SYMBOL_TABLE
"CONTROL_DAT"	DB 1	DB 1
"MODBUS_HPARAM_PN_2"	DB 2	DB 2
"CPULINDB"	DB 30	DB 30
"SYS_Date_Time_D"	DB 34	DB 34	// 系统日期和时间设置和读取数据区
"FB200_DB"	DB 200	FB 200
"FB201_DB"	DB 201	FB 201
"MAIN-READ-SLAVE"	DB 202	DB 202
"MAIN-WRITE-SLAVE"	DB 203	DB 203
"MAIN-READ-IBP"	DB 204	DB 204
"MAIN-WRITE-IBP"	DB 205	DB 205
"DETAIL_DIAG_DB_RACK0"	DB 458	FB 315	// DB FOR SFB13
"DETAIL_DIAG_DB_RACK1"	DB 459	FB 315	// DB FOR SFB12
"DP_ERROR_RACK0"	DB 460	DB 460
"DP_ERROR_RESET_DB"	DB 461	DB 461
"DP_ERROR_FB1501"	DB 462	FB 1501
"DB_FOR_FB300"	DB 463	FB 300
"DP_VAT"	DB 464	DB 464
"DP_ERROR_RACK1"	DB 465	DB 465
"DP_ERROR1_RESET"	DB 466	DB 466
"DP_ERROR1_FB1501"	DB 467	FB 1501
"FB523_DB"	DB 523	FB 523
"LED"	DB 525	DB 525
"IDB_MODBUS"	DB 915	FB 915
"JOBLIST_DB"	DB 919	FB 919
"JOB_RESET_DB"	DB 921	FB 921
"LSQK-1"	DB 2005	DB 2005
"EPS22"	DB 2015	DB 2015
"AP-PSB"	DB 2025	DB 2025
"XFSW"	DB 2035	DB 2035
"ZNZM_WRITE"	DB 2053	DB 2053
"ZNZM_READ"	DB 2055	DB 2055
"YSB_1_2"	DB 2065	DB 2065
"YSB_3_4"	DB 2075	DB 2075
"AP PSB  WSB"	DB 2115	DB 2115
"E420/04(K1)"	DB 2125	DB 2125
"E420/08(K4)"	DB 2135	DB 2135
"H420/02(K4)"	DB 2145	DB 2145
"E402\02_N RE"	DB 2185	DB 2185
"IMCC_Read"	DB 2291	DB 2291	// IMCC系统读取数据
"IMCC_Write"	DB 2292	DB 2292	// IMCC系统写数据
"HF3_EPS_HMI"	DB 2501	FB 2501	// EPS_ToHMI
"IMCC_lock"	DB 2555	DB 2555
"MAIN_HMI_SCtrl"	DB 6001	DB 6001	// HMI控制设备DB
"MAIN_ToHMI"	DB 6002	DB 6002	// 发送数据至HMI
"SLAVE_HMI_SCtrl"	DB 6003	DB 6003
"SLAVE_ToHMI"	DB 6004	DB 6004
"IBP_HMI_SCtrl"	DB 6005	DB 6005
"IBP_ToHMI"	DB 6006	DB 6006
"HF3_DP_Statu_ToHMI"	DB 6007	DB 6007
"HF3_PLC_Statu_ToHMI"	DB 6008	DB 6008
"HF4_Sum_SCtrl"	DB 6040	DB 6040
"HF3_Mode_Table"	DB 7001	DB 7001	// 下载模式总表
"HF3_Act_Mode"	DB 7002	DB 7002
"HF3_Init_Mode_Index"	DB 7003	DB 7003	// 系统模式分区索引
"HF3_Mode_DB"	DB 7004	DB 7004	// 模式内部使用DB
"Maste_To_Slave_Mod_DB"	DB 7005	DB 7005	// 从端反馈模式信息至主端
"HF3_Slave_To_Maste_Mode"	DB 7006	DB 7006	// 从端反馈模式状态
"P_RCV"	FB 12	FB 12	// Receive Data from CP340
"P_SEND"	FB 13	FB 13	// Send Data to CP340
"pid"	FB 41	FB 41
"TSEND"	FB 63	FB 63	// Send Data
"TRCV"	FB 64	FB 64	// Receive Data
"TCON"	FB 65	FB 65	// Connect
"TDISCON"	FB 66	FB 66	// Disconnect
"P_RESET"	FB 177	FB 177	// Reset Job for CP340
"S7400H-COM-MAIN-SLAVE"	FB 200	FB 200
"S7400H-COM-MAIN-IBP"	FB 201	FB 201
"READ_ERROR"	FB 300	FB 300
"DETAIL_DP_DIAG"	FB 315	FB 315
"H_STATUS"	FB 523	FB 523	// Status H-System
"HF3_ZNZM_Luxtrans"	FB 730	FB 730	// 智能照明照度转换
"TCP_COMM"	FB 913	FB 913	// TCP Kommunikation
"MOD_CLI"	FB 914	FB 914
"MB_PNHCL"	FB 915	FB 915
"Job_List"	FB 919	FB 919
"JOB_RESET"	FB 921	FB 921
"MODMAS_STEP7_CP340_L"	FB 1071	FB 1071
"com_check"	FB 1501	FB 1501
"HF3_PID_FB2005"	FB 2005	FB 2005	// PID处理功能块
"HF3_RunFaultSum"	FB 2006	FB 2006	// 运行时间故障次数统计
"HF3_EPS_FB2501"	FB 2501	FB 2501	// EPS主程序段
"HF4_EPS_FB2502"	FB 2502	FB 2502	// EPS功能块
"HF3_IMCC_CommOK_FB2512"	FB 2512	FB 2512	// IMCC心跳
"HF3_IMCC_CommOK_FB2513"	FB 2513	FB 2513
"HF3_LSQK_FB2521"	FB 2521	FB 2521	// 冷水群控程序段
"HF4_LSQK_FB2522"	FB 2522	FB 2522	// LSQK功能块
"HF3_JET_FB2531"	FB 2531	FB 2531	// 射流风机主程序端
"HF3_JET_FB2532"	FB 2532	FB 2532	// 射流风机功能块
"HF3_VRV_FB2541"	FB 2541	FB 2541	// 多联体空调主程序段
"HF3_VRV_FB2542"	FB 2542	FB 2542	// 多联体空调程序端
"HF4_SB_FB2551"	FB 2551	FB 2551	// 带控制水泵程序段
"HF4_SB_FB2552"	FB 2552	FB 2552	// 带控制水泵功能块
"HF4_3#SB_FB2561"	FB 2561	FB 2561	// 洞口水泵主程序段
"HF4_3#SB_FB2562"	FB 2562	FB 2562	// 洞口水泵功能块
"HF4_JSJYB_FB2571"	FB 2571	FB 2571	// 变频给水加压泵
"HF4_JSJYB"	FB 2572	FB 2572
"HF4_WSB_FB2581"	FB 2581	FB 2581	// 污水密闭提升
"HF4_WSB_FB2582"	FB 2582	FB 2582
"HF4_PSB_FB2591"	FB 2591	FB 2591	// 局部排水泵主程序
"HF4_PSB_FB2592"	FB 2592	FB 2592	// 排水泵DB转换
"HF4_1#PSB"	FB 2601	FB 2601
"HF4_1#PSB_FB2602"	FB 2602	FB 2602
"HF4_DT_FB2621"	FB 2621	FB 2621	// 电梯
"HF4_DT_FB2622"	FB 2622	FB 2622	// 电梯
"HF4_FT_FB2631"	FB 2631	FB 2631	// 扶梯
"HF4_FT_FB2362"	FB 2632	FB 2632
"HF3_FAS_FB2641"	FB 2641	FB 2641	// FAS主程序
"HF3_FAS_FB2642"	FB 2642	FB 2642
"HF3_FAS_COMM"	FB 2643	FB 2643	// 与FAS通讯功能块
"HF4_IMCC_TVF_FB2651"	FB 2651	FB 2651	// 隧道风机主程序段
"HF4_IMCC_TVF_FB2652"	FB 2652	FB 2652	// 隧道风机功能块
"HF4_IMCC_UOF_FB2661"	FB 2661	FB 2661	// 排热风机主程序
"HF4_IMCC_UOF_FB2662"	FB 2662	FB 2662	// 排热风机功能块
"HF4_IMCC_KT_FB2671"	FB 2671	FB 2671	// 大空调主程序
"HF4_IMCC_KT_FB2672"	FB 2672	FB 2672	// 空调机组功能块
"HF4_IMCC_HPF_FB2681"	FB 2681	FB 2681	// IMCC_HPF_主程序
"HF4_IMCC_HPF_FB2682"	FB 2682	FB 2682	// IMCC_HPF功能块
"HF4_IMCC_FJ_FB2691"	FB 2691	FB 2691	// 智能低压小风机
"HF4_IMCC_FJ_FB2692"	FB 2692	FB 2692	// 智能低压小风机功能块
"HF4_IMCC_DT_FB2711"	FB 2711	FB 2711	// IMCC风量调节阀程序
"HF4_IMCC_DT_FB2712"	FB 2712	FB 2712	// IMCC风量调节阀块
"HF4_IMCC_D_FB2721"	FB 2721	FB 2721	// IMCC电动风阀主程序
"HF4_IMCC_D_FB2722"	FB 2722	FB 2722	// IMCC电动风阀功能块
"HF4_JH_YC_FB2731"	FB 2731	FB 2731	// 电子净化压差主程序
"HF4_DPH_FB2751"	FB 2751	FB 2751	// 二通阀主程序
"HF4_DPH_FB2752"	FB 2752	FB 2752	// 二通阀主程序
"picontrol"	FB 2753	FB 2753
"HF3_FJ_FB2761"	FB 2761	FB 2761	// 高架站风机主程序段
"HF3_FJ_FB2762"	FB 2762	FB 2762	// 高架站风机
"HF4_FJPG_FB2771"	FB 2771	FB 2771	// 风机盘管主程序段
"HF4_FJPG_FB2772"	FB 2772	FB 2772	// 风机盘管功能块
"HF4_XFDF_FB2781"	FB 2781	FB 2781	// 手电一体蝶阀程序段
"HF4_XVDF_FB2782"	FB 2782	FB 2782	// 手电一体蝶阀功能块
"HF4_EPS_WLE_FB2791"	FB 2791	FB 2791	// 区间疏散指示
"HF4_EPS_WLE_FB2792"	FB 2792	FB 2792	// 区间疏散指示功能块
"HF3_D_FB2801"	FB 2801	FB 2801	// 高架站风阀主程序
"HF3_D_FB2802"	FB 2802	FB 2802	// 高架站风阀功能块
"HF4_FHF_RFM_FB2811"	FB 2811	FB 2811	// 防火阀人防门
"HF4_Senor_FB2821"	FB 2821	FB 2821	// 传感器程序段
"HF4_Sensor_FB2822"	FB 2822	FB 2822	// 传感器功能块
"AB_IBP_Comm"	FB 2831	FB 2831
"ZNZM_6biao"	FB 2841	FB 2841
"HF3_WSB_FB2852"	FB 2852	FB 2852
"HF3_Mode_Pro"	FB 3000	FB 3000	// 模式表总程序
"HF4_Mode_CAL_FB3001"	FB 3001	FB 3001
"HF3_Mode LookUp_FB3002"	FB 3002	FB 3002	// 查总模式表
"HF3_Mode_BE_Judge_FB3003"	FB 3003	FB 3003
"HF3_Sys_Grp_FB3004"	FB 3004	FB 3004	// 系统群控及状态上传
"HF3_Mode_Explode_FB3005"	FB 3005	FB 3005	// 模式表分解
"HF3_Mode_Condition_3006"	FB 3006	FB 3006
"HF3_SYS_Init"	FB 3007	FB 3007	// 系统初始化
"HF3_Slave_To_Maste"	FB 3009	FB 3009
"HF3_Mode_Refuse_FB3010"	FB 3010	FB 3010	// 模式不符合判断
"HF3_Big_LookUp_FB3012"	FB 3012	FB 3012	// 查表子程序
"HF3_Tub_LookUp_FB3013"	FB 3013	FB 3013
"HF3_little_LookUp_FB3014"	FB 3014	FB 3014
"HF3_WG_Be_Judge_FB3015"	FB 3015	FB 3015	// 判断模式开始/结束/执行中
"HF3_Sys_Grp_FB3016"	FB 3016	FB 3016
"HF3_LittleSys_Grp_FB3017"	FB 3017	FB 3017
"HF3_Mode_Condition_3018"	FB 3018	FB 3018
"HF3_Mode_Explode_FB3019"	FB 3019	FB 3019
"SDT"	FB 4180	FB 4180
"BAS_CGQ"	FB 4251	FB 4251
"IMCC_Pro"	FC 1	FC 1	// 智能低压通信数据段
"HF3_B_T_W_FC51"	FC 51	FC 51	// BOOLתWORD
"HF3_W_T_B_FC54"	FC 54	FC 54	// WORDתBOOL
"HF3_Bite_T_Bool_FC55"	FC 55	FC 55
"SCALE"	FC 105	FC 105	// Scaling Values
"UNSCALE"	FC 106	FC 106	// Unscaling Values
"MK_ERROR_SAVE_RACK0"	FC 201	FC 201
"RIO_Information"	FC 202	FC 202
"MK_ERROR_SAVE_RACK1"	FC 203	FC 203
"DP_ERROR_TO_DB701"	FC 204	FC 204
"GET_DBN"	FC 501	FC 501	// Get DB Nummer
"BAS_CLOCK"	FC 505	FC 505
"CPU_Information"	FC 523	FC 523
"HF3_ZNZM_Time_Trans"	FC 731	FC 731	// 智能照明校时
"ZNZM_CURRENT_ILLU_TRANS"	FC 732	FC 732	// 智能低压通信数据段
"ABS_I"	FC 1234	FC 1234
"real_to_int"	FC 2000	FC 2000
"HF3_IMCC_FC2511"	FC 2511	FC 2511
"HF3_LSQK_FC2821"	FC 2821	FC 2821	// 冷水机组函数
"HF3_Maste_To_Slave_Mode"	FC 3008	FC 3008	// 模式执行序列传送
"HF3_Mode_Refuse_FC3010"	FC 3010	FC 3010	// 模式不符判断
"HF4_FUZHI"	FC 4000	FC 4000
"HF3_CP340_FC4301"	FC 4301	FC 4301	// CP340_配置程序段
"A_B_IBP_Comm"	FC 4311	FC 4311	// BAS内部通讯
"XFDF_B1_LR"	I 0.0	BOOL	// 远程/就地状态
"XFDF_B1_Opd"	I 0.1	BOOL	// 开状态
"XFDF_B1_Cld"	I 0.2	BOOL	// 关状态
"XFDF_B1_GFlt"	I 0.3	BOOL	// 综合故障报警信号
"XFDF_B2_LR"	I 0.4	BOOL	// 远程/就地状态
"XFDF_B2_Opd"	I 0.5	BOOL	// 开状态
"XFDF_B2_Cld"	I 0.6	BOOL	// 关状态
"XFDF_B2_GFlt"	I 0.7	BOOL	// 综合故障报警信号
"RFM_1_opd"	I 1.0	BOOL	// 开反馈
"RFM_2_opd"	I 1.1	BOOL	// 开反馈
"SDPH_B1_LR"	I 1.2	BOOL	// 就地/远程信号
"SDPH_K1_B1_LR"	I 1.3	BOOL	// 就地/远程信号
"SDPH_K2_B1_LR"	I 1.4	BOOL	// 就地/远程信号
"SDPH_K3_B1_LR"	I 1.5	BOOL	// 就地/远程信号
"YC_B_Alarm"	I 2.0	BOOL	// 压差开关报警
"JH_B_Run"	I 2.1	BOOL	// 运行信号
"JH_B_Stp"	I 2.2	BOOL	// 停止信号
"JH_B_Wash"	I 2.3	BOOL	// 清洗信号
"JH_B_Flt"	I 2.4	BOOL	// 综合故障报警信号
"JH_B_Auto"	I 2.5	BOOL	// 自动/手动信号
"EPS12_QJSS_UEF_Opd"	I 4.0	BOOL	// 上行头前向反馈
"EPS12_QJSS_UEB_Opd"	I 4.1	BOOL	// 上行头后向反馈
"EPS12_QJSS_DHF_Opd"	I 4.2	BOOL	// 下行尾前向反馈
"EPS12_QJSS_DHB_Opd"	I 4.3	BOOL	// 下行尾后向反馈
"Always0"	M 0.0	BOOL
"Always1"	M 0.1	BOOL
"IMCC_CommOK"	M 50.0	BOOL	// 智能低压通信判断
"JOB_PLUS"	M 100.0	BOOL
"FAS_CODE"	MW 120	INT
"HF3_Main_OB1"	OB 1	OB 1	// 程序主循环
"CYC_INT5"	OB 35	OB 35	// Cyclic Interrupt 5
"RED_I/O_FLT1"	OB 70	OB 70	// Redundancy I/O Fault 1
"RED_FLT"	OB 72	OB 72	// Redundancy Fault
"PS_FLT"	OB 81	OB 81	// Power Supply Fault
"I/O_FLT1"	OB 82	OB 82	// I/O ZOint Fault 1
"I/O_FLT2"	OB 83	OB 83	// I/O Point Fault 2
"CPU_FLT"	OB 84	OB 84	// CPU Fault
"OBNL_FLT"	OB 85	OB 85	// OB Not Loaded Fault
"RACK_FLT"	OB 86	OB 86	// Loss of Rack Fault
"COMM_FLT"	OB 87	OB 87	// Communication Fault
"COMPLETE RESTART"	OB 100	OB 100	// Complete Restart
"PROG_ERR"	OB 121	OB 121	// Programming Error
"MOD_ERR"	OB 122	OB 122	// Module Access Error
"T_A1_aiHumi"	PIW 512	INT	// 湿度反馈
"T_A1_aiTemp"	PIW 514	INT	// 温度反馈
"T_B1_aiHumi"	PIW 516	INT	// 湿度反馈
"T_B1_aiTemp"	PIW 518	INT	// 温度反馈
"H_B1_aiHumi"	PIW 520	INT	// 湿度反馈
"H_B1_aiTemp"	PIW 522	INT	// 温度反馈
"H_B2_aiHumi"	PIW 524	INT	// 湿度反馈
"H_B2_aiTemp"	PIW 526	INT	// 温度反馈
"H_B3_aiHumi"	PIW 528	INT	// 湿度反馈
"H_B3_aiTemp"	PIW 530	INT	// 温度反馈
"K1_H_B1_aiHumi"	PIW 532	INT	// 湿度反馈
"K1_H_B1_aiTemp"	PIW 534	INT	// 温度反馈
"K2_H_B1_aiHumi"	PIW 536	INT	// 湿度反馈
"K2_H_B1_aiTemp"	PIW 538	INT	// 温度反馈
"K3_H_B1_aiHumi"	PIW 540	INT	// 湿度反馈
"K3_H_B1_aiTemp"	PIW 542	INT	// 温度反馈
"C_A1_aiCO2"	PIW 552	INT	// 二氧化碳浓度反馈
"C_B1_aiCO2"	PIW 554	INT	// 二氧化碳浓度反馈
"SDPH_B1_aiPFB"	PIW 560	INT	// 开度反馈
"SDPH_K1_B1_aiPFB"	PIW 562	INT	// 开度反馈
"SDPH_K2_B1_aiPFB"	PIW 564	INT	// 开度反馈
"SDPH_K3_B1_aiPFB"	PIW 566	INT	// 开度反馈
"H_B7_aiHumi"	PIW 576	INT	// 湿度反馈
"H_B7_aiTemp"	PIW 578	INT	// 温度反馈
"H_B6_aiHumi"	PIW 580	INT	// 湿度反馈
"H_B6_aiTemp"	PIW 582	INT	// 温度反馈
"T_B2_aiHumi"	PIW 584	INT	// 湿度反馈
"T_B2_aiTemp"	PIW 586	INT	// 温度反馈
"K2_T_B1_aiHumi"	PIW 588	INT	// 湿度反馈
"K2_T_B1_aiTemp"	PIW 590	INT	// 温度反馈
"K1_T_B6_aiHumi"	PIW 592	INT	// 湿度反馈
"K1_T_B6_aiTemp"	PIW 594	INT	// 温度反馈
"C_B4_aiCO2"	PIW 600	INT	// 二氧化碳浓度反馈
"C_B2_aiCO2"	PIW 602	INT	// 二氧化碳浓度反馈
"H_B5_aiHumi"	PIW 608	INT	// 湿度反馈
"H_B5_aiTemp"	PIW 610	INT	// 温度反馈
"H_B4_aiHumi"	PIW 612	INT	// 湿度反馈
"H_B4_aiTemp"	PIW 614	INT	// 温度反馈
"K1_T_B1_aiHumi"	PIW 616	INT	// 湿度反馈
"K1_T_B1_aiTemp"	PIW 618	INT	// 温度反馈
"K1_T_B2_aiHumi"	PIW 620	INT	// 湿度反馈
"K1_T_B2_aiTemp"	PIW 622	INT	// 温度反馈
"K1_T_B3_aiHumi"	PIW 624	INT	// 湿度反馈
"K1_T_B3_aiTemp"	PIW 626	INT	// 温度反馈
"K1_T_B4_aiHumi"	PIW 628	INT	// 湿度反馈
"K1_T_B4_aiTemp"	PIW 630	INT	// 温度反馈
"K1_T_B5_aiHumi"	PIW 632	INT	// 湿度反馈
"K1_T_B5_aiTemp"	PIW 634	INT	// 温度反馈
"K3_T_B1_aiHumi"	PIW 636	INT	// 湿度反馈
"K3_T_B1_aiTemp"	PIW 638	INT	// 温度反馈
"C_B3_aiCO2"	PIW 664	INT	// 二氧化碳浓度反馈
"SDPH_B_aqPset"	PQW 512	INT	// 开度控制
"SDPH_K1_B1_aqPset"	PQW 514	INT	// 开度控制
"SDPH_K2_B1_aqPset"	PQW 520	INT	// 开度控制
"SDPH_K3_B1_aqPset"	PQW 522	INT	// 开度控制
"XFDF_B1_Opn"	Q 0.0	BOOL	// 开控制
"XFDF_B1_Cls"	Q 0.1	BOOL	// 关控制
"XFDF_B2_Opn"	Q 0.2	BOOL	// 开控制
"XFDF_B2_Cls"	Q 0.3	BOOL	// 关控制
"EPS12_QJSS_UEF_opn"	Q 2.0	BOOL	// 上行头前向控制
"EPS12_QJSS_UEB_opn"	Q 2.1	BOOL	// 上行头后向控制
"EPS12_QJSS_DHF_opn"	Q 2.2	BOOL	// 下行尾前向控制
"EPS12_QJSS_DHB_opn"	Q 2.3	BOOL	// 下行尾后向控制
"TP"	SFB 3	SFB 3	// Generate a Pulse
"TON"	SFB 4	SFB 4	// Generate an On Delay
"BSEND"	SFB 12	SFB 12	// Sending Segmented Data
"BRCV"	SFB 13	SFB 13	// Receiving Segmented Data
"ALARM_8P"	SFB 35	SFB 35	// Generate Block-Related Messages with Values for 8 Signals
"RDREC"	SFB 52	SFB 52	// Read a Process Data Record
"WRREC"	SFB 53	SFB 53	// Write a Process Data Record
"READ_CLK"	SFC 1	SFC 1	// Read System Clock
"GADR_LGC"	SFC 5	SFC 5	// Query Logical Address of a Channel
"RD_SINFO"	SFC 6	SFC 6	// Read OB Start Information
"DPNRM_DG"	SFC 13	SFC 13	// Read Diagnostic Data of a DP Slave
"BLKMOV"	SFC 20	SFC 20	// Copy Variables
"TEST_DB"	SFC 24	SFC 24	// Test Data Block
"DIS_AIRT"	SFC 41	SFC 41	// Delay the Higher Priority Interrupts and Asynchronous Errors
"EN_AIRT"	SFC 42	SFC 42	// Enable Higher Priority Interrupts and Asynchronous Errors
"LGC_GADR"	SFC 49	SFC 49	// Query the Module Slot Belonging to a Logical Address
"RDSYSST"	SFC 51	SFC 51	// Read a System Status List or Partial List
"WR_REC"	SFC 58	SFC 58	// Write Data Record
"RD_REC"	SFC 59	SFC 59	// Read a Data Record
"T800"	T 800	TIMER
"UDT_ANY_Pointer"	UDT 10	UDT 10
"VAT_1"	VAT 1	
"VAT_2_LSQK"	VAT 2	
"ZNZM_TEST"	VAT 3	
"VAT_sctrl"	VAT 4	
"VAT_DB2292"	VAT 5	
"Client_Job"	VAT 6	
END_SYMBOL_TABLE
